Staubli VAL3: get.pgx

public program get(string& x_sItem[], num x_nIndex)
begin
  x_sItem=right(listCall[x_nIndex],len(listCall[x_nIndex])-1)
end
